{attribute 'GeneratedUsingTerminal: EL2521-0000-1017'}
{attribute addProperty BoxType "EL2521-0000-1017"}
{attribute addProperty Id "Frequency_selectBOOL1Disable_rampBOOL1Go_counterBOOL1"}
{attribute addProperty CRC "3673038162"}
{attribute addProperty Size "3"}
TYPE Control_DAEE1D52 :
STRUCT
	{attribute addProperty Name "Frequency_select"}
	Frequency_select : BOOL;
	{attribute addProperty Name "Disable_ramp"}
	Disable_ramp : BOOL;
	{attribute addProperty Name "Go_counter"}
	Go_counter : BOOL;
END_STRUCT
END_TYPE

(* stored: Version 1.2.0.0, ProductVersion 3.1.4024.9
   DUT Control_DAEE1D52: Id {85783818-13e5-4bea-9e0c-5a80cec8c1ec} *)
